TYPE ST_MC :
STRUCT
	Power 			: Tc2_MC2.MC_POWER;
	MoveAbsolute 	: Tc2_MC2.MC_MoveAbsolute;	
	MoveRelative 	: Tc2_MC2.MC_MoveRelative;
END_STRUCT
END_TYPE

(* stored: Version 1.1.0.1, ProductVersion 3.1.4024.12
   DUT ST_MC: Id {e87bf896-9231-4520-a679-e6ae0efc462e} *)
